PROGRAM AxisJog
VAR
	lrJogSpeed	: POINTER TO LREAL;
END_VAR

// 快速Jog速度设定
IF bJogFast THEN
	lrJogSpeed := ADR(aAxis_Jog_Speed[1]);
ELSE
	lrJogSpeed := ADR(aAxis_Jog_Speed[0]);
END_IF


IF bManualCtrl_Part_LeftArm_Left THEN

	axis_LeftArm_Left_Jog(
		Axis:= axis_LeftArm_Left, 
		JogForward:= bAxis_LeftArm_Left_JogP , 			// 如果想ABS的时候按下JOG按键不停止ABS动作就加上后面的判断AND NOT axis_LeftArm_Left_MoveAbs.Active
		JogBackwards:= bAxis_LeftArm_Left_JogN, 		// 如果想ABS的时候按下JOG按键不停止ABS动作就加上后面的判断AND NOT axis_LeftArm_Left_MoveAbs.Active
		Mode:= MC_JOGMODE_CONTINOUS, 					//需要设置为MC_JOGMODE_CONTINOUS下面的速度设定才有效
		Position:= , 
		Velocity:= lrJogSpeed^, 
		Acceleration:= , 
		Deceleration:= , 
		Jerk:= , 
		Done=> , 
		Busy=> , 
		Active=> , 
		CommandAborted=> , 
		Error=> , 
		ErrorID=> );

END_IF

END_PROGRAM

(* stored: Version 1.1.0.1, ProductVersion 3.1.4024.14
   POU AxisJog: Id {74d5a483-6847-47e3-a03b-541646338622}, SpecialFunc None *)
